// TIA Portal V16 export
// export: Created 2021-11-12T13:31:55.8851385Z, ExportSetting WithDefaults, DisplayName Totally Integrated Automation Portal, DisplayVersion V16 Update 3, DisplayName TIA Portal Version Control Interface, DisplayVersion V16 Update 2, DisplayName TIA Portal Openness, DisplayVersion V16 Update 3, DisplayName SINAMICS Startdrive Advanced, DisplayVersion V16 Update 5, DisplayName SINAMICS Startdrive G130, G150, S120, S150, SINAMICS MV, S210, DisplayVersion V16 Update 5, DisplayName SINAMICS Startdrive G110M, G120, G120C, G120D, G120P, G115D, DisplayVersion V16 Update 5, DisplayName STEP 7 Professional, DisplayVersion V16 Update 3, DisplayName STEP 7 Safety, DisplayVersion V16, DisplayName WinCC UA Professional, DisplayVersion V16 Update 3
DATA_BLOCK "IDB_Cab_000+UC10_DB"   // DB214
VERSION : 0.1
// stored: AutoNumber true, DBAccessibleFromOPCUA true, InstanceOfName Cab_000+UC10, InstanceOfType FB
"Cab_000+UC10"
   // VAR
   //    "SF_UC10-FV01_11_Alarm" { S7_SetPoint := 'True'} : "STD_DI_Mon";
   //    "SF_UC10-FB21_14_Alarm" { S7_SetPoint := 'True'} : "STD_DI_Mon";
   //    "SF_UC10-FC21_14_Alarm" { S7_SetPoint := 'True'} : "STD_DI_Mon";
   //    "SF_UC10-EC01_3_Alarm" { S7_SetPoint := 'True'} : "STD_DI_Mon";
   //    "SF_UC10-FC01_14_Alarm" { S7_SetPoint := 'True'} : "STD_DI_Mon";
   //    "SF_UC10-TB01_14_Alarm" { S7_SetPoint := 'True'} : "STD_DI_Mon";
   //    "SF_UC10-FC30_14_Alarm" { S7_SetPoint := 'True'} : "STD_DI_Mon";
   //    "SF_UC10-FC30_24_Alarm" { S7_SetPoint := 'True'} : "STD_DI_Mon";
   //    "SF_UC10-FC50_14_Alarm" { S7_SetPoint := 'True'} : "STD_DI_Mon";
   //    "SF_UC10-FC51_24_Alarm" { S7_SetPoint := 'True'} : "STD_DI_Mon";
   //    "SF_UC12-FC21_14_Alarm" { S7_SetPoint := 'True'} : "STD_DI_Mon";
   //    "SF_UC12-EC01_3_Alarm" { S7_SetPoint := 'True'} : "STD_DI_Mon";
   //    "SF_UC11-FC01_14_Alarm" { S7_SetPoint := 'True'} : "STD_DI_Mon";
   //    "SF_UC11-FC02_14_Alarm" { S7_SetPoint := 'True'} : "STD_DI_Mon";
   //    "SF_UC11-FC03_14_Alarm" { S7_SetPoint := 'True'} : "STD_DI_Mon";
   // END_VAR
BEGIN
END_DATA_BLOCK
